// TIA Portal V19 export
VAR_GLOBAL   // PLC tag table "LB112"
   LB112_Decoiler_Lp_Bwd AT %Q116.3 : Bool;   // 324SH6
   LB112_Decoiler_Lp_Fwd AT %Q116.2 : Bool;   // 324SH5
   LB112_Decoiler_Pb_Bwd AT %I118.7 : Bool;   // 324SH6
   LB112_Decoiler_Pb_Fwd AT %I118.6 : Bool;   // 324SH5
   LB112_Peeler_Lp_Bwd AT %Q115.5 : Bool;   // 323SH6
   LB112_Peeler_Lp_Down AT %Q115.3 : Bool;   // 323SH4
   LB112_Peeler_Lp_Fwd AT %Q115.4 : Bool;   // 323SH5
   LB112_Peeler_Lp_Up AT %Q115.2 : Bool;   // 323SH3
   LB112_Peeler_Pb_Bwd AT %I118.1 : Bool;   // 323SH6
   LB112_Peeler_Pb_Down AT %I117.7 : Bool;   // 323SH4
   LB112_Peeler_Pb_Fwd AT %I118.0 : Bool;   // 323SH5
   LB112_Peeler_Pb_Up AT %I117.6 : Bool;   // 323SH3
   LB112_Snubber_Lp_Bwd AT %Q116.1 : Bool;   // 324SH4
   LB112_Snubber_Lp_Down AT %Q115.7 : Bool;   // 324SH2
   LB112_Snubber_Lp_Fwd AT %Q116.0 : Bool;   // 324SH3
   LB112_Snubber_Lp_Up AT %Q115.6 : Bool;   // 324SH1
   LB112_Snubber_Pb_Bwd AT %I118.5 : Bool;   // 324SH4
   LB112_Snubber_Pb_Down AT %I118.3 : Bool;   // 324SH2
   LB112_Snubber_Pb_Fwd AT %I118.4 : Bool;   // 324SH3
   LB112_Snubber_Pb_Up AT %I118.2 : Bool;   // 324SH1
   LB112_Straightener_Lp_Bwd AT %Q115.1 : Bool;   // 323SH2
   LB112_Straightener_Lp_Fwd AT %Q115.0 : Bool;   // 323SH1
   LB112_Straightener_Pb_Bwd AT %I117.5 : Bool;   // 323SH2
   LB112_Straightener_Pb_Fwd AT %I117.4 : Bool;   // 323SH1
   LB112_Straightener_Sel_Close AT %I117.3 : Bool;   // 323SA1
   LB112_Straightener_Sel_Open AT %I117.2 : Bool;   // 323SA1
   LB112_Button_L AT %I1034.1 : Bool;   // 104DI1 - 200SB1
   LB112_Button_R AT %I1034.5 : Bool;   // 104DI5 - 200SB2
END_VAR
